// TwinCAT 3 PLC project AnalogSensors
// ProgramVersion: 3.1.4023.0
// libraries:
//   Tc2_SerialCom, * (Beckhoff Automation GmbH)
//   Tc2_Standard, * (Beckhoff Automation GmbH)
//   Tc2_System, * (Beckhoff Automation GmbH)
//   Tc3_Module, * (Beckhoff Automation GmbH)
// project tree:
//   GVLs/ MyGVL.TcGVL, SensorValues.TcGVL
//   / PlcTask.TcTTO
//   POUs/ FB_CO2Sensor.TcPOU, FB_InteriorOperationMonitoring.TcPOU, FB_PressureSensor.TcPOU, FB_HumiditySensor.TcPOU, MAIN.TcPOU (not stored), FB_TemperatureSensor.TcPOU
// real-time tasks:
//   TASK PlcTask: cycle T#10ms, priority 20, ADS port 350
//   TASK PlcTask1: cycle T#10ms, priority 21, ADS port 351
// I/O:
//   DEVICE Gerät 1 (EtherCAT), AmsNetId 10.183.66.136.2.1
//     Klemme 2 (EK1100) [EK1100 EtherCAT-Koppler (2A E-Bus)]
//       Klemme 3 (EL3208-0010) [EL3208-0010 8K. Ana. Eingang PT1000 (RTD)]
//       Klemme 4 (EL9011) [EL9011 Endklemme]
// variable links:
//   AnalogSensors/AnalogSensors Instance <-> Device 1 (EtherCAT)/Term 2 (EK1100)/Term 3 (EL3208-0010)
//     PlcTask Inputs/MyGVL.iInput1 <-> RTD Inputs Channel 1/Value

CONFIGURATION AnalogSensors
    RESOURCE PLC ON TwinCAT3
        TASK PlcTask(INTERVAL := T#10ms, PRIORITY := 21);
        PROGRAM MAIN WITH PlcTask : MAIN;
    END_RESOURCE
END_CONFIGURATION

// ---- GVLs/MyGVL.TcGVL
{attribute 'qualified_only'}
VAR_GLOBAL
	iInput1 AT %I* : INT;
END_VAR

// ---- GVLs/SensorValues.TcGVL
{attribute 'qualified_only'}
VAR_GLOBAL
	rCO2Value AT %Q* : REAL;
	rPressure AT %Q* : REAL;
	rHumidity AT %Q* : REAL;
	rTemperature AT %Q* : REAL;
END_VAR

// ---- POUs/FB_CO2Sensor.TcPOU
FUNCTION_BLOCK FB_CO2Sensor
VAR_INPUT
END_VAR
VAR_OUTPUT
END_VAR
VAR
	rCO2Value : REAL;
	iRange : INT := 32767;
	iVmax : INT := 10;
	iCorrespondenceFactor : INT := 1000;
END_VAR

rCO2Value := (INT_TO_REAL(MyGVL.iInput1)/iRange)*iVmax * iCorrespondenceFactor;

PROPERTY getCO2Value : REAL
GET
getCO2Value := rCO2Value;
END_GET
END_PROPERTY

END_FUNCTION_BLOCK

// ---- POUs/FB_InteriorOperationMonitoring.TcPOU
FUNCTION_BLOCK FB_InteriorOperationMonitoring
VAR_INPUT
END_VAR
VAR_OUTPUT
END_VAR
VAR
	fb_humiditysensor : FB_HumiditySensor;
	fb_cO2sensor : FB_CO2Sensor;
	fb_temperaturesensor : FB_TemperatureSensor;
	fb_pressuresensor : FB_PressureSensor;
END_VAR

METHOD updateSensorValues
VAR_INPUT
END_VAR
fb_cO2sensor();
fb_humiditysensor();
fb_pressuresensor();
fb_temperaturesensor();

SensorValues.rCO2Value := fb_cO2sensor.getCO2Value;
SensorValues.rHumidity := fb_humiditysensor.getHumidity;
SensorValues.rPressure := fb_pressuresensor.getPressure;
SensorValues.rTemperature := fb_temperaturesensor.getTemperature;
END_METHOD

END_FUNCTION_BLOCK

// ---- POUs/FB_HumiditySensor.TcPOU
FUNCTION_BLOCK FB_HumiditySensor
VAR_INPUT
END_VAR
VAR_OUTPUT
END_VAR
VAR
	rHumidity : REAL;
	iRange : INT := 32767;
	iVmax : INT := 10;
	rZeroOffset : REAL := 0.95800;
	rSlope : REAL := 0.03068;
END_VAR

rHumidity := ((INT_TO_REAL(MyGVL.iInput1)/iRange)*iVmax - rZeroOffset)/rSlope;

PROPERTY getHumidity : REAL
GET
getHumidity := rHumidity;
END_GET
END_PROPERTY

END_FUNCTION_BLOCK

// ---- POUs/FB_TemperatureSensor.TcPOU
FUNCTION_BLOCK FB_TemperatureSensor
VAR_INPUT
END_VAR
VAR_OUTPUT
END_VAR
VAR
	rTemperature : REAL;
	rCorrespondenceFactor : REAL := 0.01;
END_VAR

rTemperature := INT_TO_REAL(MyGVL.iInput1) * rCorrespondenceFactor;

PROPERTY getTemperature : REAL
GET
getTemperature := rTemperature;
END_GET
END_PROPERTY

END_FUNCTION_BLOCK

// ---- POUs/FB_PressureSensor.TcPOU
FUNCTION_BLOCK FB_PressureSensor
VAR_INPUT
END_VAR
VAR_OUTPUT
END_VAR
VAR
	rPressure : REAL;
END_VAR

PROPERTY getPressure : REAL
GET
getPressure := rPressure;
END_GET
END_PROPERTY

END_FUNCTION_BLOCK
